SYSTEM DASDAass2_t (* System Configuration *)
  (* Standard: 61499-1 *)
  (* Version 0.4, 2009-03-05, JHC, Holobloc Inc., Deleted Application. *)
  (* Version 0.3, 2003-12-05, JHC, Rockwell Automation, Renamed from NEWSYSTEM. *)
  (* Version 0.2, 2002-11-05, JHC, Rockwell Automation, Fixed missing (empty) FBD in Application. *)
  (* Version 0.1, 2002-01-17, JHC, Rockwell Automation, Minor cleanup *)
  (* Version 0.0, 2000-05-27, JHC, Rockwell Automation *)
  DEVICE HMI_LAYER : FRAME_DEVICE(BOUNDS := [0,0,200,400])
    RESOURCE HMI_1 : PANEL_RESOURCE(COLS := 1, ROWS := 0)
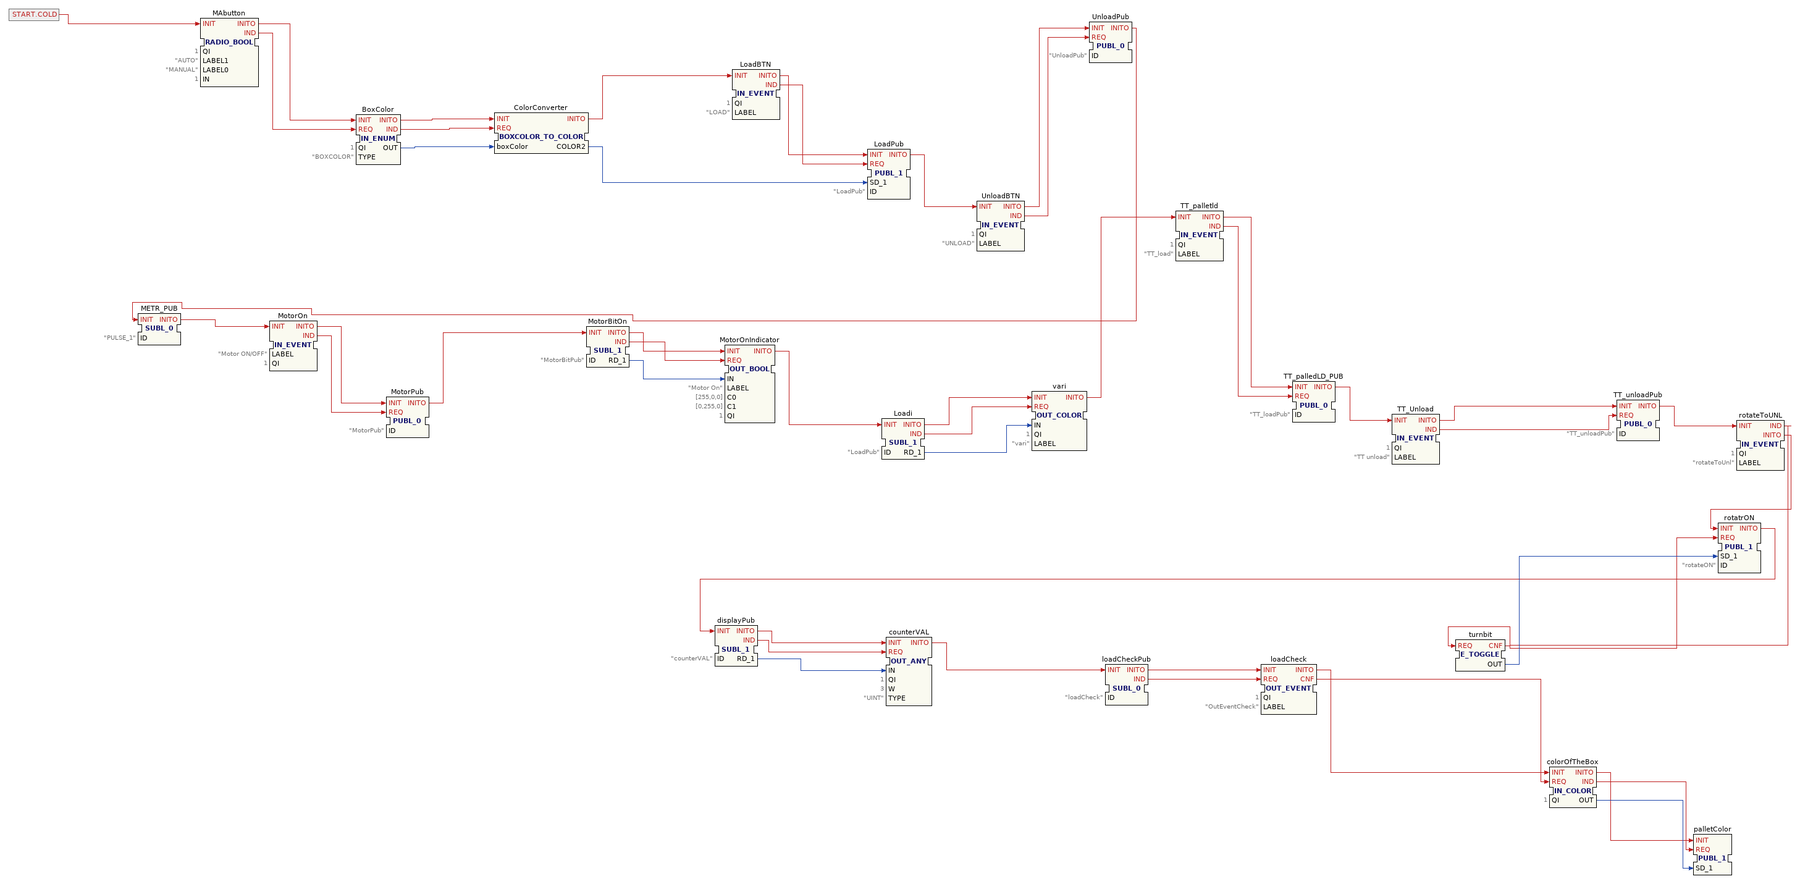
      FBS
        MAbutton : RADIO_BOOL(QI := 1, LABEL1 := "AUTO", LABEL0 := "MANUAL", IN := 1);
        LoadPub : PUBL_1(ID := "LoadPub");
        ColorConverter : BOXCOLOR_TO_COLOR;
        BoxColor : IN_ENUM(QI := 1, TYPE := "BOXCOLOR");
        LoadBTN : IN_EVENT(QI := 1, LABEL := "LOAD");
        Loadi : SUBL_1(ID := "LoadPub");
        vari : OUT_COLOR(QI := 1, LABEL := "vari");
        METR_PUB : SUBL_0(ID := "PULSE_1");
        MotorOn : IN_EVENT(LABEL := "Motor ON/OFF", QI := 1);
        MotorPub : PUBL_0(ID := "MotorPub");
        MotorBitOn : SUBL_1(ID := "MotorBitPub");
        MotorOnIndicator : OUT_BOOL(LABEL := "Motor On", C0 := [255,0,0], C1 := [0,255,0], QI := 1);
        UnloadBTN : IN_EVENT(QI := 1, LABEL := "UNLOAD");
        UnloadPub : PUBL_0(ID := "UnloadPub");
        TT_palletld : IN_EVENT(QI := 1, LABEL := "TT_load");
        TT_palledLD_PUB : PUBL_0(ID := "TT_loadPub");
        displayPub : SUBL_1(ID := "counterVAL");
        counterVAL : OUT_ANY(QI := 1, W := 3, TYPE := "UINT");
        loadCheckPub : SUBL_0(ID := "loadCheck");
        loadCheck : OUT_EVENT(QI := 1, LABEL := "OutEventCheck");
        rotateToUNL : IN_EVENT(QI := 1, LABEL := "rotateToUnl");
        turnbit : E_TOGGLE;
        rotatrON : PUBL_1(ID := "rotateON");
        TT_Unload : IN_EVENT(QI := 1, LABEL := "TT unload");
        TT_unloadPub : PUBL_0(ID := "TT_unloadPub");
        colorOfTheBox : IN_COLOR(QI := 1);
        palletColor : PUBL_1;
      END_FBS
      EVENT_CONNECTIONS
        START.COLD TO MAbutton.INIT;
        BoxColor.INITO TO ColorConverter.INIT;
        BoxColor.IND TO ColorConverter.REQ;
        MAbutton.INITO TO BoxColor.INIT;
        MAbutton.IND TO BoxColor.REQ;
        ColorConverter.INITO TO LoadBTN.INIT;
        LoadBTN.INITO TO LoadPub.INIT;
        LoadBTN.IND TO LoadPub.REQ;
        Loadi.INITO TO vari.INIT;
        Loadi.IND TO vari.REQ;
        METR_PUB.INITO TO MotorOn.INIT;
        MotorOn.INITO TO MotorPub.INIT;
        MotorOn.IND TO MotorPub.REQ;
        MotorPub.INITO TO MotorBitOn.INIT;
        MotorBitOn.INITO TO MotorOnIndicator.INIT;
        MotorBitOn.IND TO MotorOnIndicator.REQ;
        LoadPub.INITO TO UnloadBTN.INIT;
        UnloadBTN.INITO TO UnloadPub.INIT;
        UnloadBTN.IND TO UnloadPub.REQ;
        MotorOnIndicator.INITO TO Loadi.INIT;
        UnloadPub.INITO TO METR_PUB.INIT;
        TT_palletld.INITO TO TT_palledLD_PUB.INIT;
        TT_palletld.IND TO TT_palledLD_PUB.REQ;
        vari.INITO TO TT_palletld.INIT;
        displayPub.INITO TO counterVAL.INIT;
        displayPub.IND TO counterVAL.REQ;
        counterVAL.INITO TO loadCheckPub.INIT;
        loadCheckPub.INITO TO loadCheck.INIT;
        loadCheckPub.IND TO loadCheck.REQ;
        rotateToUNL.IND TO turnbit.REQ;
        rotateToUNL.INITO TO rotatrON.INIT;
        rotatrON.INITO TO displayPub.INIT;
        turnbit.CNF TO rotatrON.REQ;
        TT_palledLD_PUB.INITO TO TT_Unload.INIT;
        TT_Unload.INITO TO TT_unloadPub.INIT;
        TT_unloadPub.INITO TO rotateToUNL.INIT;
        TT_Unload.IND TO TT_unloadPub.REQ;
        loadCheck.INITO TO colorOfTheBox.INIT;
        loadCheck.CNF TO colorOfTheBox.REQ;
        colorOfTheBox.INITO TO palletColor.INIT;
        colorOfTheBox.IND TO palletColor.REQ;
      END_CONNECTIONS
      DATA_CONNECTIONS
        BoxColor.OUT TO ColorConverter.boxColor;
        ColorConverter.COLOR2 TO LoadPub.SD_1;
        Loadi.RD_1 TO vari.IN;
        MotorBitOn.RD_1 TO MotorOnIndicator.IN;
        displayPub.RD_1 TO counterVAL.IN;
        turnbit.OUT TO rotatrON.SD_1;
        colorOfTheBox.OUT TO palletColor.SD_1;
      END_CONNECTIONS
    END_RESOURCE
  END_DEVICE
  DEVICE VIEW_LAYER : FRAME_DEVICE(BOUNDS := [250,0,900,900])
    RESOURCE VIEW_RES : VIEW_PANEL(DIA := 85, SIZE := [10,8], VERTICAL := 0)
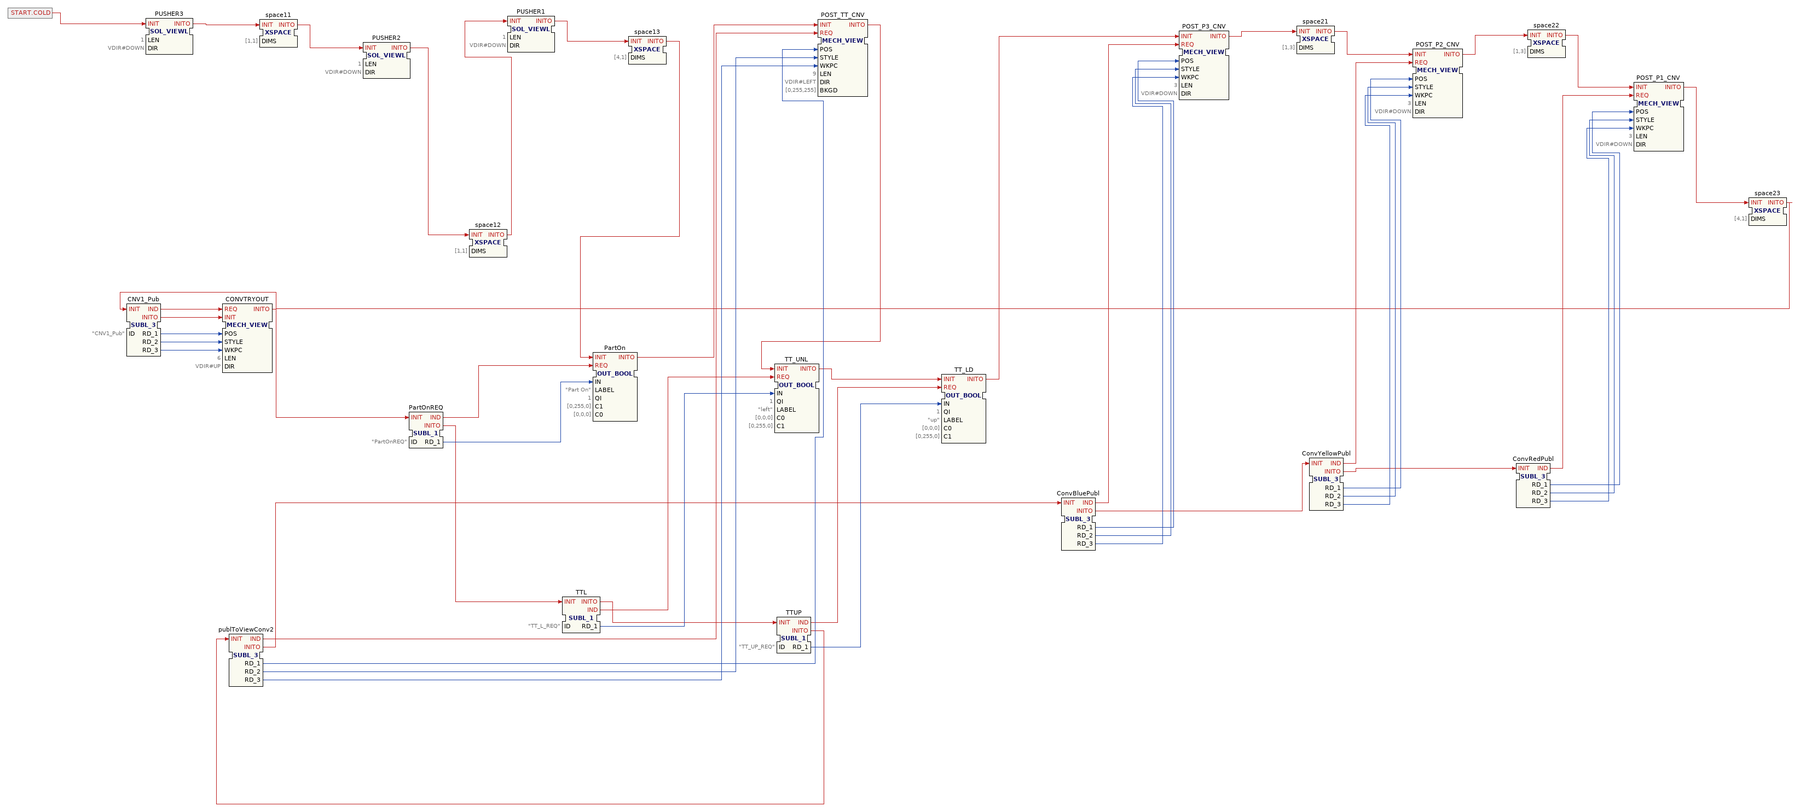
      FBS
        PUSHER3 : SOL_VIEWL(LEN := 1, DIR := VDIR#DOWN);
        space11 : XSPACE(DIMS := [1,1]);
        PUSHER2 : SOL_VIEWL(LEN := 1, DIR := VDIR#DOWN);
        space12 : XSPACE(DIMS := [1,1]);
        PUSHER1 : SOL_VIEWL(LEN := 1, DIR := VDIR#DOWN);
        space13 : XSPACE(DIMS := [4,1]);
        space21 : XSPACE(DIMS := [1,3]);
        space22 : XSPACE(DIMS := [1,3]);
        space23 : XSPACE(DIMS := [4,1]);
        POST_P1_CNV : MECH_VIEW(LEN := 3, DIR := VDIR#DOWN);
        POST_P2_CNV : MECH_VIEW(LEN := 3, DIR := VDIR#DOWN);
        POST_P3_CNV : MECH_VIEW(LEN := 3, DIR := VDIR#DOWN);
        POST_TT_CNV : MECH_VIEW(LEN := 9, DIR := VDIR#LEFT, BKGD := [0,255,255]);
        CONVTRYOUT : MECH_VIEW(LEN := 6, DIR := VDIR#UP);
        CNV1_Pub : SUBL_3(ID := "CNV1_Pub");
        PartOnREQ : SUBL_1(ID := "PartOnREQ");
        PartOn : OUT_BOOL(LABEL := "Part On", QI := 1, C1 := [0,255,0], C0 := [0,0,0]);
        TT_UNL : OUT_BOOL(QI := 1, LABEL := "left", C0 := [0,0,0], C1 := [0,255,0]);
        TT_LD : OUT_BOOL(QI := 1, LABEL := "up", C0 := [0,0,0], C1 := [0,255,0]);
        TTL : SUBL_1(ID := "TT_L_REQ");
        TTUP : SUBL_1(ID := "TT_UP_REQ");
        publToViewConv2 : SUBL_3;
        ConvRedPubl : SUBL_3;
        ConvYellowPubl : SUBL_3;
        ConvBluePubl : SUBL_3;
      END_FBS
      EVENT_CONNECTIONS
        START.COLD TO PUSHER3.INIT;
        PUSHER3.INITO TO space11.INIT;
        space11.INITO TO PUSHER2.INIT;
        PUSHER2.INITO TO space12.INIT;
        space12.INITO TO PUSHER1.INIT;
        PUSHER1.INITO TO space13.INIT;
        space22.INITO TO POST_P1_CNV.INIT;
        POST_P1_CNV.INITO TO space23.INIT;
        space21.INITO TO POST_P2_CNV.INIT;
        POST_P2_CNV.INITO TO space22.INIT;
        POST_P3_CNV.INITO TO space21.INIT;
        CNV1_Pub.IND TO CONVTRYOUT.REQ;
        space23.INITO TO CNV1_Pub.INIT;
        CNV1_Pub.INITO TO CONVTRYOUT.INIT;
        CONVTRYOUT.INITO TO PartOnREQ.INIT;
        space13.INITO TO PartOn.INIT;
        PartOn.INITO TO POST_TT_CNV.INIT;
        PartOnREQ.IND TO PartOn.REQ;
        POST_TT_CNV.INITO TO TT_UNL.INIT;
        TT_UNL.INITO TO TT_LD.INIT;
        TT_LD.INITO TO POST_P3_CNV.INIT;
        PartOnREQ.INITO TO TTL.INIT;
        TTL.INITO TO TTUP.INIT;
        TTL.IND TO TT_UNL.REQ;
        TTUP.IND TO TT_LD.REQ;
        TTUP.INITO TO publToViewConv2.INIT;
        publToViewConv2.IND TO POST_TT_CNV.REQ;
        ConvRedPubl.IND TO POST_P1_CNV.REQ;
        ConvYellowPubl.IND TO POST_P2_CNV.REQ;
        ConvBluePubl.IND TO POST_P3_CNV.REQ;
        publToViewConv2.INITO TO ConvBluePubl.INIT;
        ConvBluePubl.INITO TO ConvYellowPubl.INIT;
        ConvYellowPubl.INITO TO ConvRedPubl.INIT;
      END_CONNECTIONS
      DATA_CONNECTIONS
        CNV1_Pub.RD_1 TO CONVTRYOUT.POS;
        CNV1_Pub.RD_2 TO CONVTRYOUT.STYLE;
        CNV1_Pub.RD_3 TO CONVTRYOUT.WKPC;
        PartOnREQ.RD_1 TO PartOn.IN;
        TTL.RD_1 TO TT_UNL.IN;
        TTUP.RD_1 TO TT_LD.IN;
        publToViewConv2.RD_1 TO POST_TT_CNV.POS;
        publToViewConv2.RD_2 TO POST_TT_CNV.STYLE;
        publToViewConv2.RD_3 TO POST_TT_CNV.WKPC;
        ConvRedPubl.RD_1 TO POST_P1_CNV.POS;
        ConvRedPubl.RD_2 TO POST_P1_CNV.STYLE;
        ConvRedPubl.RD_3 TO POST_P1_CNV.WKPC;
        ConvYellowPubl.RD_1 TO POST_P2_CNV.POS;
        ConvYellowPubl.RD_2 TO POST_P2_CNV.STYLE;
        ConvYellowPubl.RD_3 TO POST_P2_CNV.WKPC;
        ConvBluePubl.RD_1 TO POST_P3_CNV.POS;
        ConvBluePubl.RD_2 TO POST_P3_CNV.STYLE;
        ConvBluePubl.RD_3 TO POST_P3_CNV.WKPC;
      END_CONNECTIONS
    END_RESOURCE
  END_DEVICE
  DEVICE MODEL_LAYER : FRAME_DEVICE
    RESOURCE INIT_CLOCK : PANEL_RESOURCE
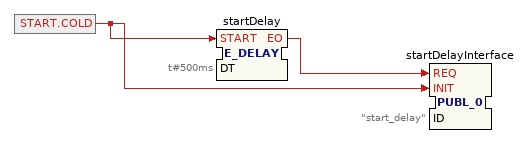
      FBS
        startDelay : E_DELAY(DT := t#500ms);
        startDelayInterface : PUBL_0(ID := "start_delay");
      END_FBS
      EVENT_CONNECTIONS
        START.COLD TO startDelay.START;
        startDelay.EO TO startDelayInterface.REQ;
        START.COLD TO startDelayInterface.INIT;
      END_CONNECTIONS
    END_RESOURCE
    RESOURCE MODEL_CLOCK : PANEL_RESOURCE
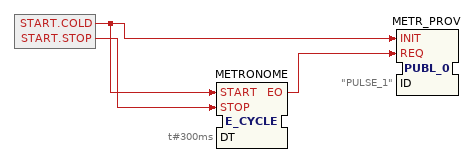
      FBS
        METRONOME : E_CYCLE(DT := t#300ms);
        METR_PROV : PUBL_0(ID := "PULSE_1");
      END_FBS
      EVENT_CONNECTIONS
        START.COLD TO METRONOME.START;
        START.STOP TO METRONOME.STOP;
        START.COLD TO METR_PROV.INIT;
        METRONOME.EO TO METR_PROV.REQ;
      END_CONNECTIONS
    END_RESOURCE
    RESOURCE CNV_1_MODEL : PANEL_RESOURCE
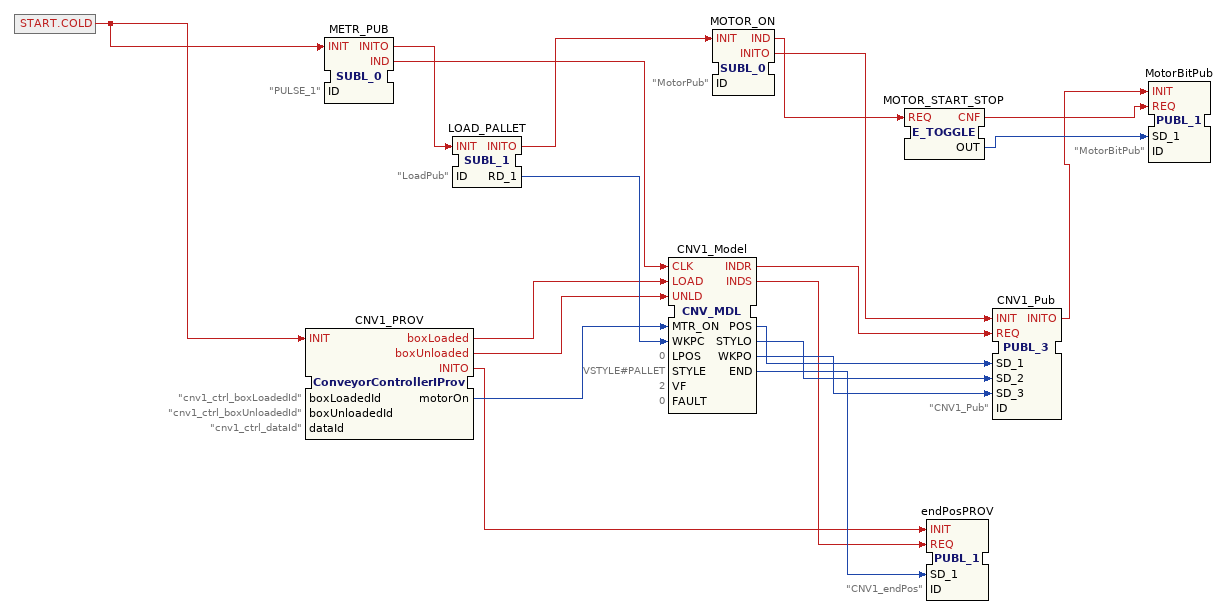
      FBS
        METR_PUB : SUBL_0(ID := "PULSE_1");
        MOTOR_ON : SUBL_0(ID := "MotorPub");
        LOAD_PALLET : SUBL_1(ID := "LoadPub");
        MOTOR_START_STOP : E_TOGGLE;
        CNV1_Model : CNV_MDL(LPOS := 0, STYLE := VSTYLE#PALLET, VF := 2, FAULT := 0);
        CNV1_Pub : PUBL_3(ID := "CNV1_Pub");
        MotorBitPub : PUBL_1(ID := "MotorBitPub");
        endPosPROV : PUBL_1(ID := "CNV1_endPos");
        CNV1_PROV : ConveyorControllerIProv(boxLoadedId := "cnv1_ctrl_boxLoadedId", boxUnloadedId := "cnv1_ctrl_boxUnloadedId", dataId := "cnv1_ctrl_dataId");
      END_FBS
      EVENT_CONNECTIONS
        START.COLD TO METR_PUB.INIT;
        METR_PUB.INITO TO LOAD_PALLET.INIT;
        LOAD_PALLET.INITO TO MOTOR_ON.INIT;
        MOTOR_ON.IND TO MOTOR_START_STOP.REQ;
        METR_PUB.IND TO CNV1_Model.CLK;
        MOTOR_ON.INITO TO CNV1_Pub.INIT;
        CNV1_Model.INDR TO CNV1_Pub.REQ;
        CNV1_Pub.INITO TO MotorBitPub.INIT;
        MOTOR_START_STOP.CNF TO MotorBitPub.REQ;
        CNV1_PROV.boxLoaded TO CNV1_Model.LOAD;
        CNV1_PROV.boxUnloaded TO CNV1_Model.UNLD;
        START.COLD TO CNV1_PROV.INIT;
        CNV1_PROV.INITO TO endPosPROV.INIT;
        CNV1_Model.INDS TO endPosPROV.REQ;
      END_CONNECTIONS
      DATA_CONNECTIONS
        CNV1_Model.POS TO CNV1_Pub.SD_1;
        CNV1_Model.STYLO TO CNV1_Pub.SD_2;
        CNV1_Model.WKPO TO CNV1_Pub.SD_3;
        MOTOR_START_STOP.OUT TO MotorBitPub.SD_1;
        CNV1_Model.END TO endPosPROV.SD_1;
        CNV1_PROV.motorOn TO CNV1_Model.MTR_ON;
        LOAD_PALLET.RD_1 TO CNV1_Model.WKPC;
      END_CONNECTIONS
    END_RESOURCE
    RESOURCE TT_MODEL : PANEL_RESOURCE
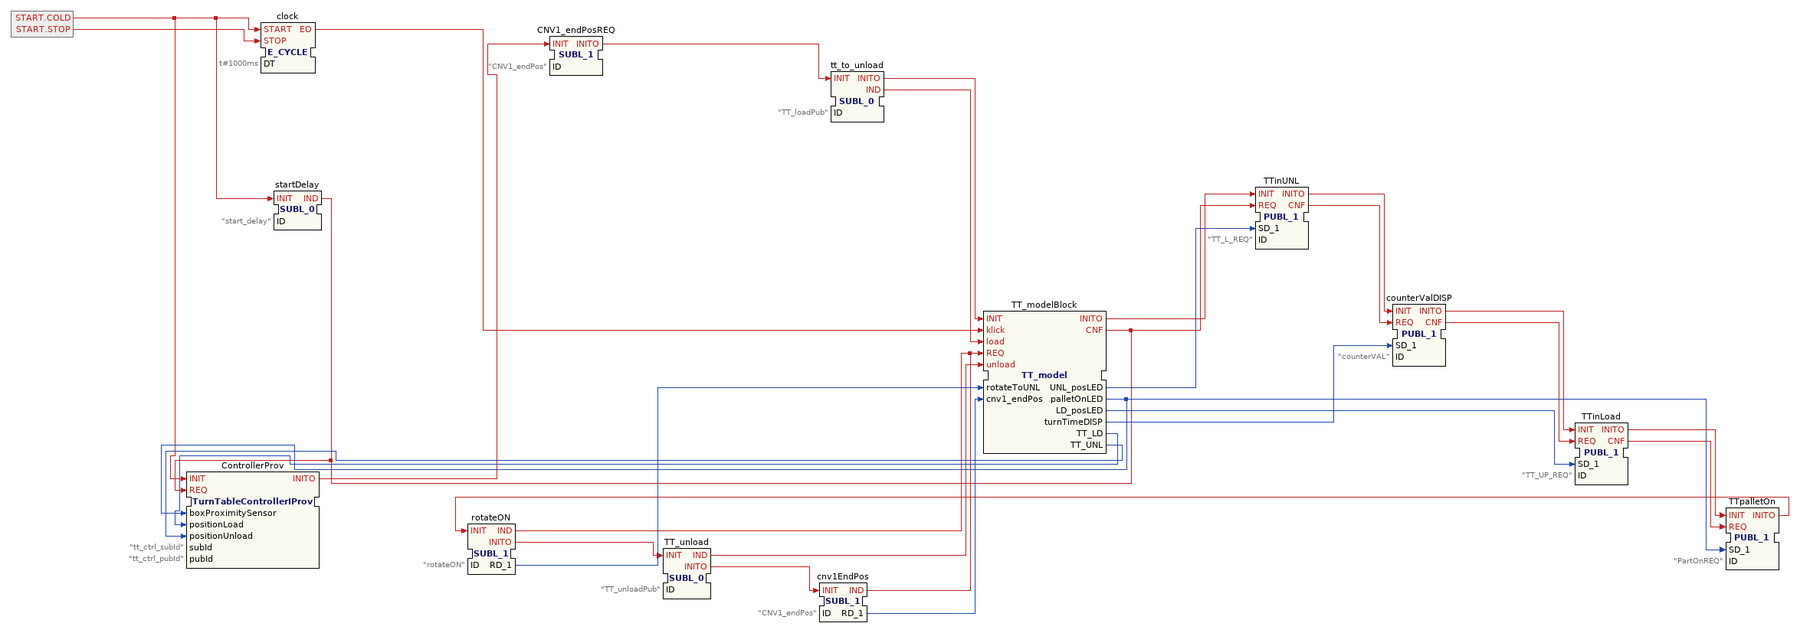
      FBS
        CNV1_endPosREQ : SUBL_1(ID := "CNV1_endPos");
        clock : E_CYCLE(DT := t#1000ms);
        ControllerProv : TurnTableControllerIProv(subId := "tt_ctrl_subId", pubId := "tt_ctrl_pubId");
        TTinUNL : PUBL_1(ID := "TT_L_REQ");
        tt_to_unload : SUBL_0(ID := "TT_loadPub");
        counterValDISP : PUBL_1(ID := "counterVAL");
        TTinLoad : PUBL_1(ID := "TT_UP_REQ");
        TTpalletOn : PUBL_1(ID := "PartOnREQ");
        rotateON : SUBL_1(ID := "rotateON");
        TT_modelBlock : TT_model;
        TT_unload : SUBL_0(ID := "TT_unloadPub");
        startDelay : SUBL_0(ID := "start_delay");
        cnv1EndPos : SUBL_1(ID := "CNV1_endPos");
      END_FBS
      EVENT_CONNECTIONS
        START.COLD TO clock.START;
        START.STOP TO clock.STOP;
        START.COLD TO ControllerProv.INIT;
        ControllerProv.INITO TO CNV1_endPosREQ.INIT;
        CNV1_endPosREQ.INITO TO tt_to_unload.INIT;
        TTinUNL.INITO TO counterValDISP.INIT;
        TTinUNL.CNF TO counterValDISP.REQ;
        counterValDISP.INITO TO TTinLoad.INIT;
        counterValDISP.CNF TO TTinLoad.REQ;
        TTinLoad.INITO TO TTpalletOn.INIT;
        TTinLoad.CNF TO TTpalletOn.REQ;
        TTpalletOn.INITO TO rotateON.INIT;
        tt_to_unload.INITO TO TT_modelBlock.INIT;
        TT_modelBlock.INITO TO TTinUNL.INIT;
        TT_modelBlock.CNF TO TTinUNL.REQ;
        clock.EO TO TT_modelBlock.klick;
        tt_to_unload.IND TO TT_modelBlock.load;
        rotateON.IND TO TT_modelBlock.REQ;
        rotateON.INITO TO TT_unload.INIT;
        TT_unload.IND TO TT_modelBlock.unload;
        START.COLD TO startDelay.INIT;
        startDelay.IND TO ControllerProv.REQ;
        TT_modelBlock.CNF TO ControllerProv.REQ;
        TT_unload.INITO TO cnv1EndPos.INIT;
        cnv1EndPos.IND TO TT_modelBlock.REQ;
      END_CONNECTIONS
      DATA_CONNECTIONS
        TT_modelBlock.UNL_posLED TO TTinUNL.SD_1;
        TT_modelBlock.palletOnLED TO TTpalletOn.SD_1;
        TT_modelBlock.LD_posLED TO TTinLoad.SD_1;
        TT_modelBlock.turnTimeDISP TO counterValDISP.SD_1;
        TT_modelBlock.palletOnLED TO ControllerProv.boxProximitySensor;
        rotateON.RD_1 TO TT_modelBlock.rotateToUNL;
        TT_modelBlock.TT_LD TO ControllerProv.positionLoad;
        TT_modelBlock.TT_UNL TO ControllerProv.positionUnload;
        cnv1EndPos.RD_1 TO TT_modelBlock.cnv1_endPos;
      END_CONNECTIONS
    END_RESOURCE
    RESOURCE CNV_2_MODEL : PANEL_RESOURCE
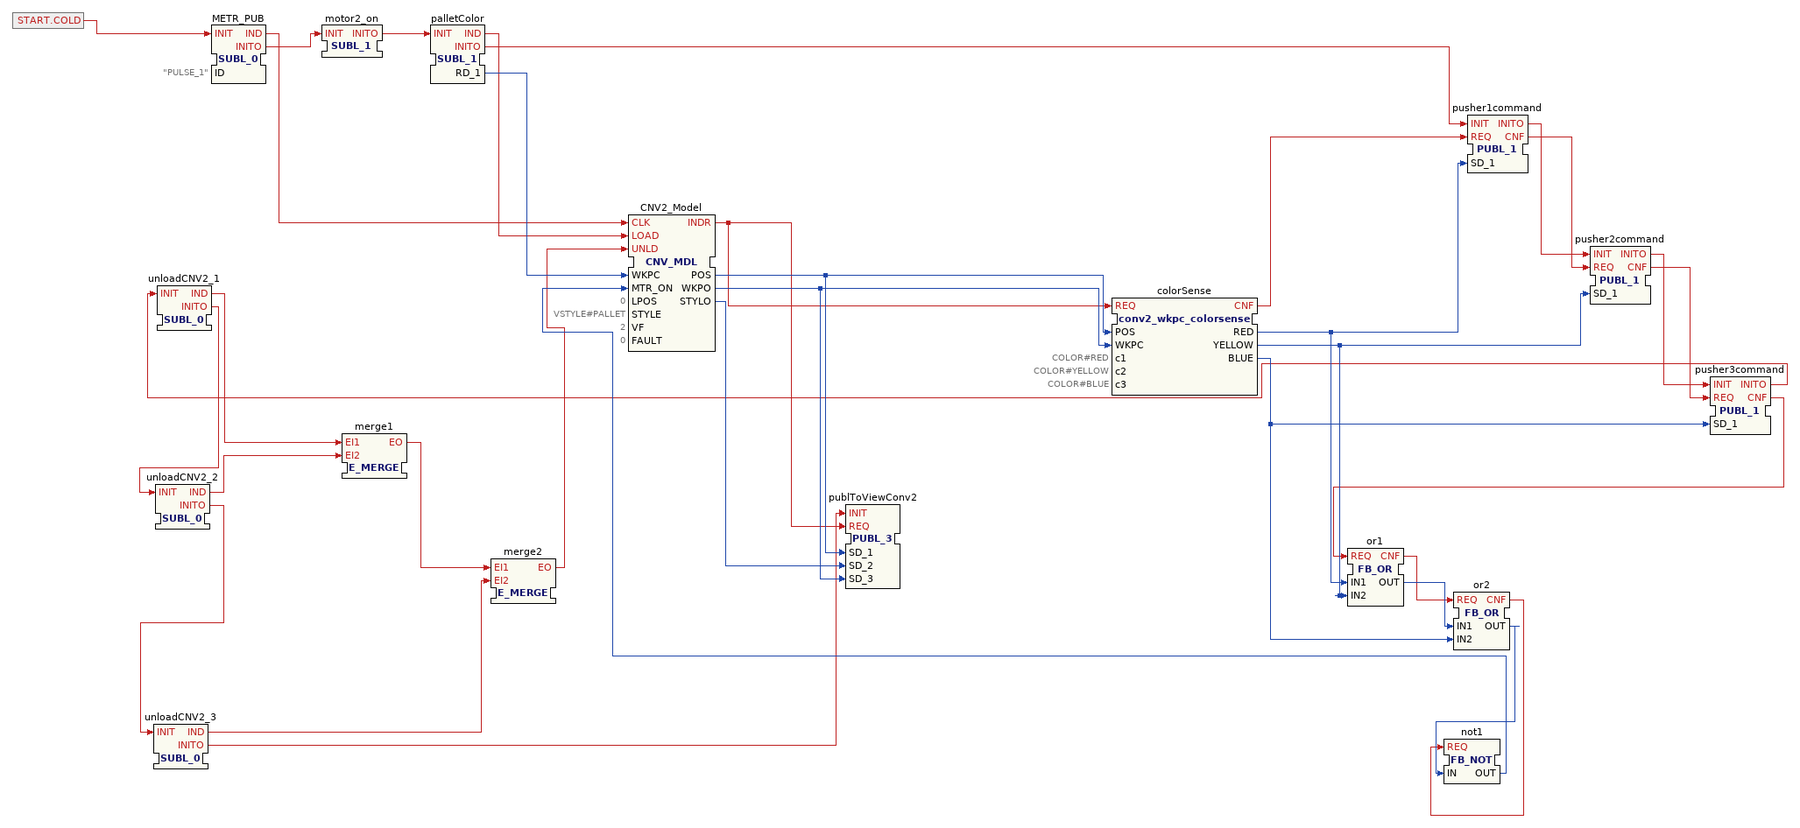
      FBS
        CNV2_Model : CNV_MDL(LPOS := 0, STYLE := VSTYLE#PALLET, VF := 2, FAULT := 0);
        METR_PUB : SUBL_0(ID := "PULSE_1");
        palletColor : SUBL_1;
        motor2_on : SUBL_1;
        colorSense : conv2_wkpc_colorsense(c1 := COLOR#RED, c2 := COLOR#YELLOW, c3 := COLOR#BLUE);
        pusher1command : PUBL_1;
        pusher2command : PUBL_1;
        pusher3command : PUBL_1;
        unloadCNV2_1 : SUBL_0;
        merge1 : E_MERGE;
        merge2 : E_MERGE;
        unloadCNV2_2 : SUBL_0;
        unloadCNV2_3 : SUBL_0;
        or1 : FB_OR;
        or2 : FB_OR;
        not1 : FB_NOT;
        publToViewConv2 : PUBL_3;
      END_FBS
      EVENT_CONNECTIONS
        START.COLD TO METR_PUB.INIT;
        METR_PUB.IND TO CNV2_Model.CLK;
        palletColor.IND TO CNV2_Model.LOAD;
        METR_PUB.INITO TO motor2_on.INIT;
        motor2_on.INITO TO palletColor.INIT;
        palletColor.INITO TO pusher1command.INIT;
        pusher1command.INITO TO pusher2command.INIT;
        pusher2command.INITO TO pusher3command.INIT;
        colorSense.CNF TO pusher1command.REQ;
        pusher1command.CNF TO pusher2command.REQ;
        pusher2command.CNF TO pusher3command.REQ;
        pusher3command.INITO TO unloadCNV2_1.INIT;
        unloadCNV2_1.IND TO merge1.EI1;
        merge1.EO TO merge2.EI1;
        unloadCNV2_1.INITO TO unloadCNV2_2.INIT;
        unloadCNV2_2.IND TO merge1.EI2;
        unloadCNV2_2.INITO TO unloadCNV2_3.INIT;
        unloadCNV2_3.IND TO merge2.EI2;
        merge2.EO TO CNV2_Model.UNLD;
        pusher3command.CNF TO or1.REQ;
        or1.CNF TO or2.REQ;
        or2.CNF TO not1.REQ;
        unloadCNV2_3.INITO TO publToViewConv2.INIT;
        CNV2_Model.INDR TO publToViewConv2.REQ;
        CNV2_Model.INDR TO colorSense.REQ;
      END_CONNECTIONS
      DATA_CONNECTIONS
        palletColor.RD_1 TO CNV2_Model.WKPC;
        CNV2_Model.POS TO colorSense.POS;
        CNV2_Model.WKPO TO colorSense.WKPC;
        colorSense.RED TO pusher1command.SD_1;
        colorSense.YELLOW TO pusher2command.SD_1;
        colorSense.BLUE TO pusher3command.SD_1;
        colorSense.RED TO or1.IN1;
        colorSense.YELLOW TO or1.IN2;
        or1.OUT TO or2.IN1;
        colorSense.BLUE TO or2.IN2;
        or2.OUT TO not1.IN;
        not1.OUT TO CNV2_Model.MTR_ON;
        CNV2_Model.POS TO publToViewConv2.SD_1;
        CNV2_Model.STYLO TO publToViewConv2.SD_2;
        CNV2_Model.WKPO TO publToViewConv2.SD_3;
      END_CONNECTIONS
    END_RESOURCE
    RESOURCE PUSHER1_MODEL : PANEL_RESOURCE
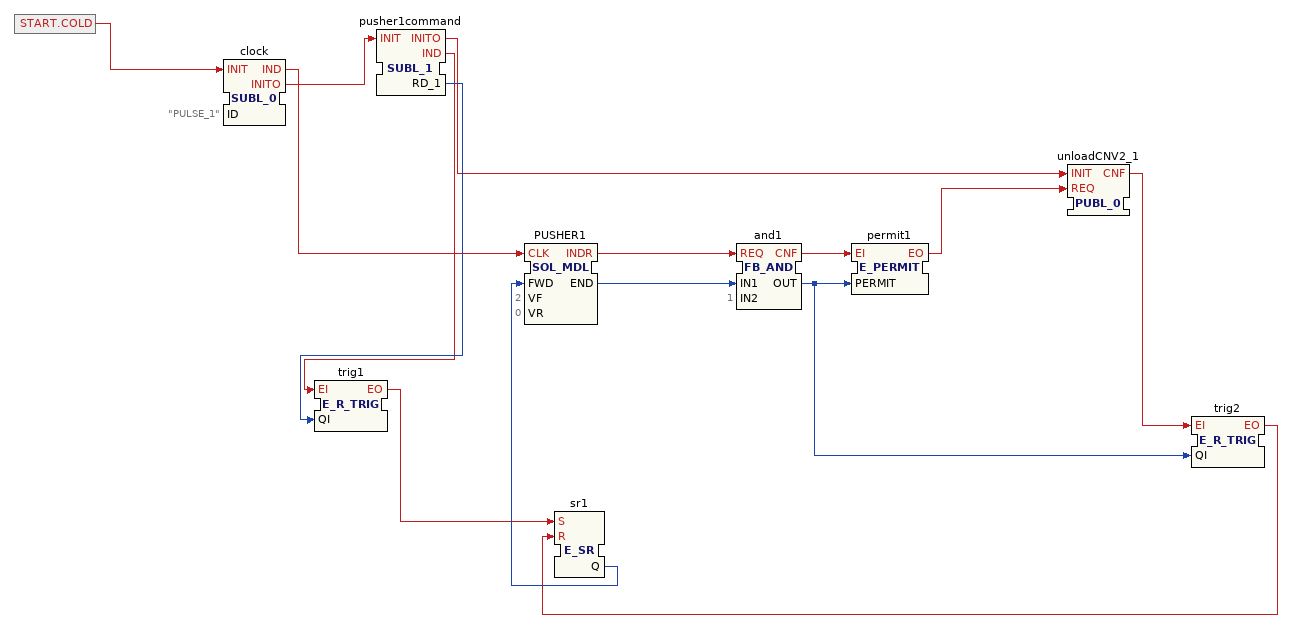
      FBS
        PUSHER1 : SOL_MDL(VF := 2, VR := 0);
        clock : SUBL_0(ID := "PULSE_1");
        pusher1command : SUBL_1;
        and1 : FB_AND(IN2 := 1);
        permit1 : E_PERMIT;
        unloadCNV2_1 : PUBL_0;
        trig1 : E_R_TRIG;
        trig2 : E_R_TRIG;
        sr1 : E_SR;
      END_FBS
      EVENT_CONNECTIONS
        START.COLD TO clock.INIT;
        clock.IND TO PUSHER1.CLK;
        clock.INITO TO pusher1command.INIT;
        PUSHER1.INDR TO and1.REQ;
        and1.CNF TO permit1.EI;
        pusher1command.INITO TO unloadCNV2_1.INIT;
        permit1.EO TO unloadCNV2_1.REQ;
        unloadCNV2_1.CNF TO trig2.EI;
        pusher1command.IND TO trig1.EI;
        trig1.EO TO sr1.S;
        trig2.EO TO sr1.R;
      END_CONNECTIONS
      DATA_CONNECTIONS
        PUSHER1.END TO and1.IN1;
        and1.OUT TO permit1.PERMIT;
        pusher1command.RD_1 TO trig1.QI;
        and1.OUT TO trig2.QI;
        sr1.Q TO PUSHER1.FWD;
      END_CONNECTIONS
    END_RESOURCE
    RESOURCE PUSHER2_MODEL : PANEL_RESOURCE
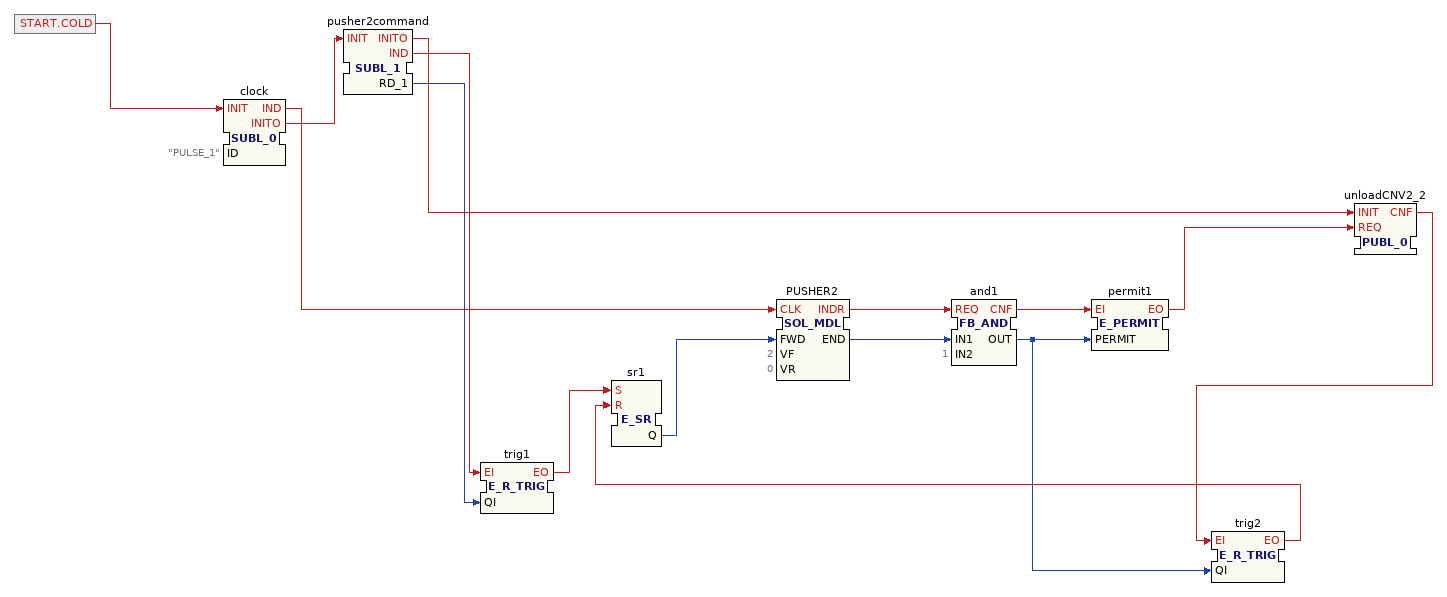
      FBS
        PUSHER2 : SOL_MDL(VF := 2, VR := 0);
        clock : SUBL_0(ID := "PULSE_1");
        pusher2command : SUBL_1;
        and1 : FB_AND(IN2 := 1);
        permit1 : E_PERMIT;
        unloadCNV2_2 : PUBL_0;
        sr1 : E_SR;
        trig1 : E_R_TRIG;
        trig2 : E_R_TRIG;
      END_FBS
      EVENT_CONNECTIONS
        START.COLD TO clock.INIT;
        clock.IND TO PUSHER2.CLK;
        clock.INITO TO pusher2command.INIT;
        PUSHER2.INDR TO and1.REQ;
        and1.CNF TO permit1.EI;
        pusher2command.INITO TO unloadCNV2_2.INIT;
        permit1.EO TO unloadCNV2_2.REQ;
        pusher2command.IND TO trig1.EI;
        trig1.EO TO sr1.S;
        unloadCNV2_2.CNF TO trig2.EI;
        trig2.EO TO sr1.R;
      END_CONNECTIONS
      DATA_CONNECTIONS
        PUSHER2.END TO and1.IN1;
        and1.OUT TO permit1.PERMIT;
        pusher2command.RD_1 TO trig1.QI;
        and1.OUT TO trig2.QI;
        sr1.Q TO PUSHER2.FWD;
      END_CONNECTIONS
    END_RESOURCE
    RESOURCE PUSHER3_MODEL : PANEL_RESOURCE
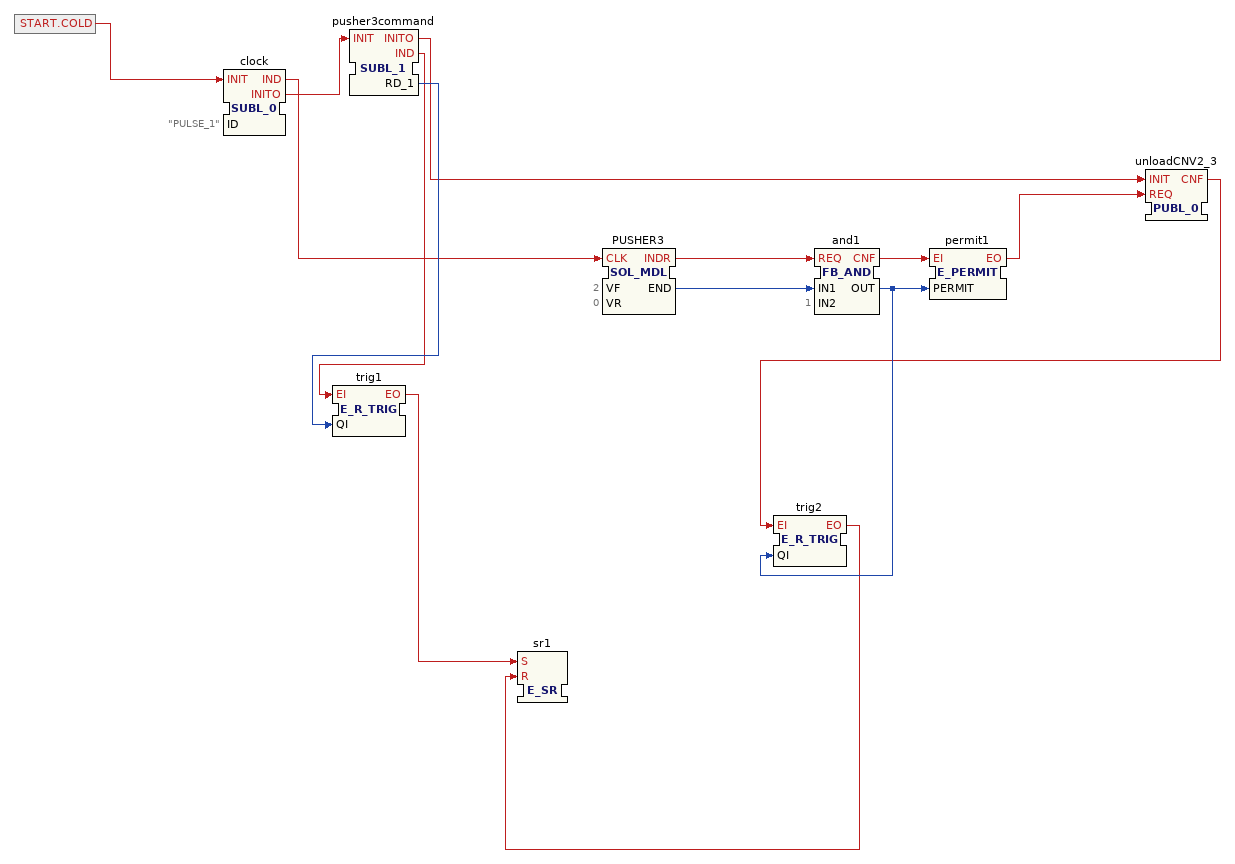
      FBS
        PUSHER3 : SOL_MDL(VF := 2, VR := 0);
        clock : SUBL_0(ID := "PULSE_1");
        pusher3command : SUBL_1;
        and1 : FB_AND(IN2 := 1);
        permit1 : E_PERMIT;
        unloadCNV2_3 : PUBL_0;
        trig1 : E_R_TRIG;
        trig2 : E_R_TRIG;
        sr1 : E_SR;
      END_FBS
      EVENT_CONNECTIONS
        START.COLD TO clock.INIT;
        clock.IND TO PUSHER3.CLK;
        clock.INITO TO pusher3command.INIT;
        PUSHER3.INDR TO and1.REQ;
        and1.CNF TO permit1.EI;
        pusher3command.INITO TO unloadCNV2_3.INIT;
        permit1.EO TO unloadCNV2_3.REQ;
        pusher3command.IND TO trig1.EI;
        trig1.EO TO sr1.S;
        unloadCNV2_3.CNF TO trig2.EI;
        trig2.EO TO sr1.R;
      END_CONNECTIONS
      DATA_CONNECTIONS
        PUSHER3.END TO and1.IN1;
        and1.OUT TO permit1.PERMIT;
        pusher3command.RD_1 TO trig1.QI;
        and1.OUT TO trig2.QI;
      END_CONNECTIONS
    END_RESOURCE
    RESOURCE CONVred_MODEL : PANEL_RESOURCE
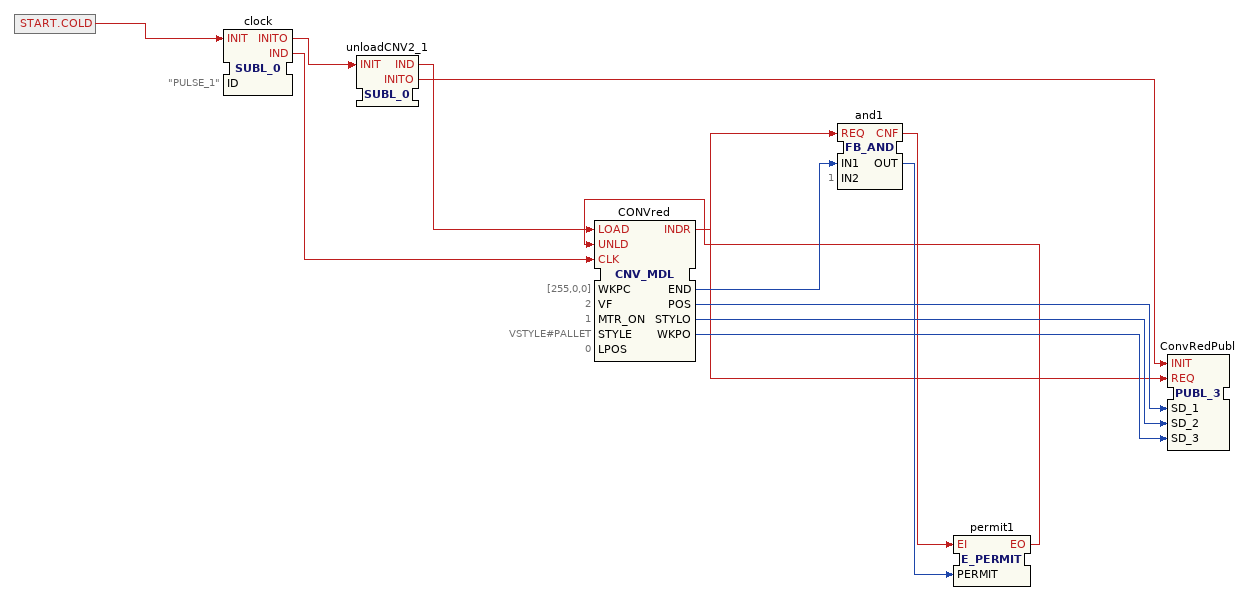
      FBS
        unloadCNV2_1 : SUBL_0;
        CONVred : CNV_MDL(WKPC := [255,0,0], VF := 2, MTR_ON := 1, STYLE := VSTYLE#PALLET, LPOS := 0);
        and1 : FB_AND(IN2 := 1);
        permit1 : E_PERMIT;
        ConvRedPubl : PUBL_3;
        clock : SUBL_0(ID := "PULSE_1");
      END_FBS
      EVENT_CONNECTIONS
        unloadCNV2_1.IND TO CONVred.LOAD;
        and1.CNF TO permit1.EI;
        permit1.EO TO CONVred.UNLD;
        unloadCNV2_1.INITO TO ConvRedPubl.INIT;
        CONVred.INDR TO ConvRedPubl.REQ;
        START.COLD TO clock.INIT;
        clock.INITO TO unloadCNV2_1.INIT;
        clock.IND TO CONVred.CLK;
        CONVred.INDR TO and1.REQ;
      END_CONNECTIONS
      DATA_CONNECTIONS
        CONVred.END TO and1.IN1;
        and1.OUT TO permit1.PERMIT;
        CONVred.POS TO ConvRedPubl.SD_1;
        CONVred.STYLO TO ConvRedPubl.SD_2;
        CONVred.WKPO TO ConvRedPubl.SD_3;
      END_CONNECTIONS
    END_RESOURCE
    RESOURCE CONVyellow_MODEL : PANEL_RESOURCE
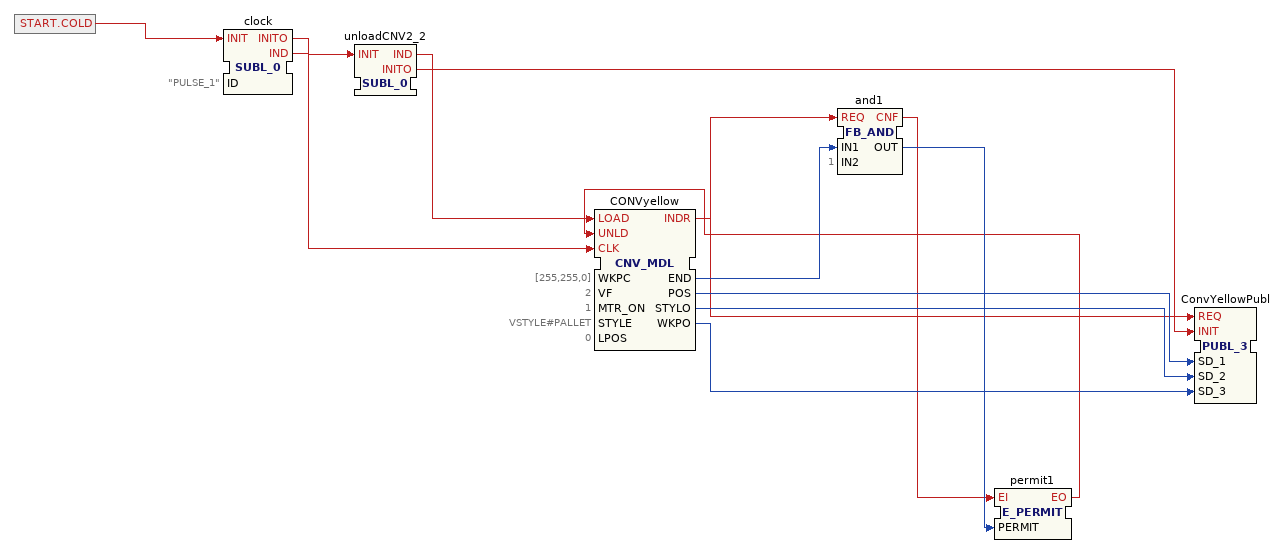
      FBS
        unloadCNV2_2 : SUBL_0;
        CONVyellow : CNV_MDL(WKPC := [255,255,0], VF := 2, MTR_ON := 1, STYLE := VSTYLE#PALLET, LPOS := 0);
        and1 : FB_AND(IN2 := 1);
        permit1 : E_PERMIT;
        ConvYellowPubl : PUBL_3;
        clock : SUBL_0(ID := "PULSE_1");
      END_FBS
      EVENT_CONNECTIONS
        unloadCNV2_2.IND TO CONVyellow.LOAD;
        and1.CNF TO permit1.EI;
        permit1.EO TO CONVyellow.UNLD;
        CONVyellow.INDR TO ConvYellowPubl.REQ;
        unloadCNV2_2.INITO TO ConvYellowPubl.INIT;
        START.COLD TO clock.INIT;
        clock.INITO TO unloadCNV2_2.INIT;
        clock.IND TO CONVyellow.CLK;
        CONVyellow.INDR TO and1.REQ;
      END_CONNECTIONS
      DATA_CONNECTIONS
        CONVyellow.END TO and1.IN1;
        and1.OUT TO permit1.PERMIT;
        CONVyellow.POS TO ConvYellowPubl.SD_1;
        CONVyellow.STYLO TO ConvYellowPubl.SD_2;
        CONVyellow.WKPO TO ConvYellowPubl.SD_3;
      END_CONNECTIONS
    END_RESOURCE
    RESOURCE CONVblue_MODEL : PANEL_RESOURCE
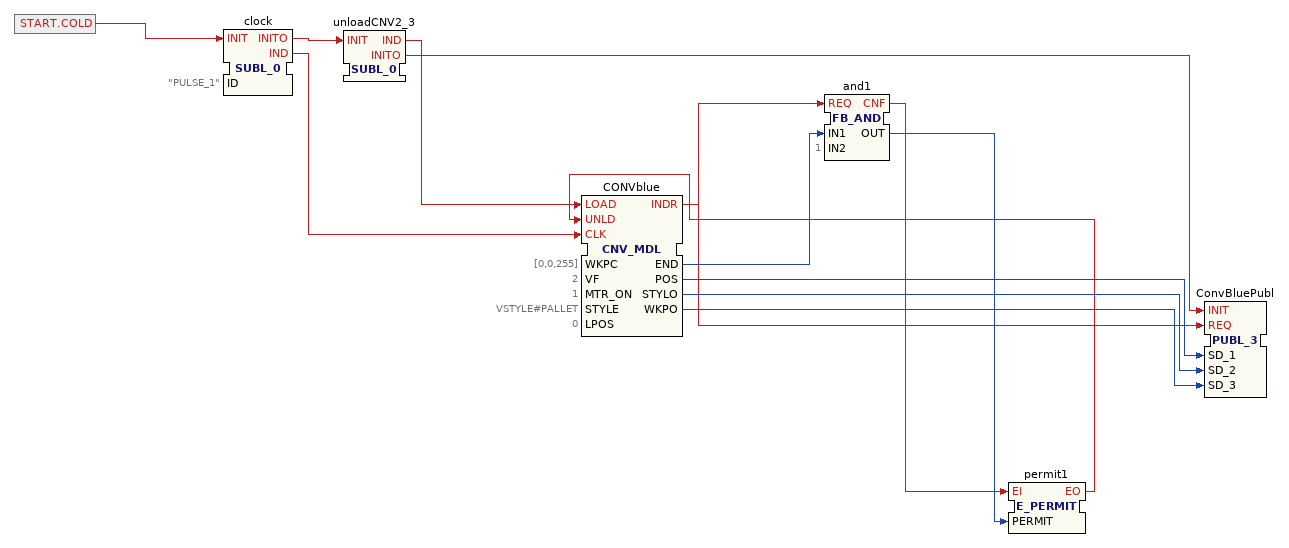
      FBS
        unloadCNV2_3 : SUBL_0;
        CONVblue : CNV_MDL(WKPC := [0,0,255], VF := 2, MTR_ON := 1, STYLE := VSTYLE#PALLET, LPOS := 0);
        and1 : FB_AND(IN2 := 1);
        permit1 : E_PERMIT;
        ConvBluePubl : PUBL_3;
        clock : SUBL_0(ID := "PULSE_1");
      END_FBS
      EVENT_CONNECTIONS
        unloadCNV2_3.IND TO CONVblue.LOAD;
        and1.CNF TO permit1.EI;
        permit1.EO TO CONVblue.UNLD;
        unloadCNV2_3.INITO TO ConvBluePubl.INIT;
        CONVblue.INDR TO ConvBluePubl.REQ;
        START.COLD TO clock.INIT;
        clock.INITO TO unloadCNV2_3.INIT;
        clock.IND TO CONVblue.CLK;
        CONVblue.INDR TO and1.REQ;
      END_CONNECTIONS
      DATA_CONNECTIONS
        CONVblue.END TO and1.IN1;
        and1.OUT TO permit1.PERMIT;
        CONVblue.POS TO ConvBluePubl.SD_1;
        CONVblue.STYLO TO ConvBluePubl.SD_2;
        CONVblue.WKPO TO ConvBluePubl.SD_3;
      END_CONNECTIONS
    END_RESOURCE
  END_DEVICE
  DEVICE CONTROLLER_LAYER : FRAME_DEVICE(BOUNDS := [0,400,200,200])
    RESOURCE Conveyor1Controller : PANEL_RESOURCE(ROWS := 0, COLS := 1)
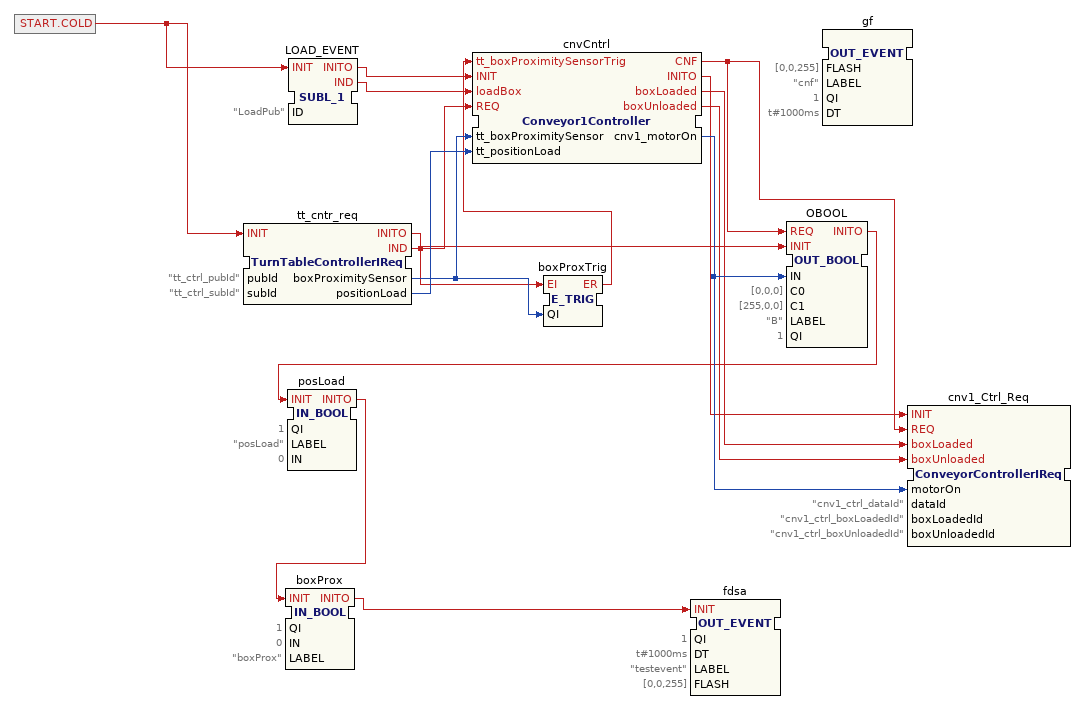
      FBS
        OBOOL : OUT_BOOL(C0 := [0,0,0], C1 := [255,0,0], LABEL := "B", QI := 1);
        gf : OUT_EVENT(FLASH := [0,0,255], LABEL := "cnf", QI := 1, DT := t#1000ms);
        cnvCntrl : Conveyor1Controller;
        boxProxTrig : E_TRIG;
        fdsa : OUT_EVENT(QI := 1, DT := t#1000ms, LABEL := "testevent", FLASH := [0,0,255]);
        posLoad : IN_BOOL(QI := 1, LABEL := "posLoad", IN := 0);
        boxProx : IN_BOOL(QI := 1, IN := 0, LABEL := "boxProx");
        cnv1_Ctrl_Req : ConveyorControllerIReq(dataId := "cnv1_ctrl_dataId", boxLoadedId := "cnv1_ctrl_boxLoadedId", boxUnloadedId := "cnv1_ctrl_boxUnloadedId");
        LOAD_EVENT : SUBL_1(ID := "LoadPub");
        tt_cntr_req : TurnTableControllerIReq(pubId := "tt_ctrl_pubId", subId := "tt_ctrl_subId");
      END_FBS
      EVENT_CONNECTIONS
        cnvCntrl.CNF TO OBOOL.REQ;
        posLoad.INITO TO boxProx.INIT;
        boxProx.INITO TO fdsa.INIT;
        boxProxTrig.ER TO cnvCntrl.tt_boxProximitySensorTrig;
        cnvCntrl.INITO TO cnv1_Ctrl_Req.INIT;
        cnvCntrl.CNF TO cnv1_Ctrl_Req.REQ;
        cnvCntrl.boxLoaded TO cnv1_Ctrl_Req.boxLoaded;
        cnvCntrl.boxUnloaded TO cnv1_Ctrl_Req.boxUnloaded;
        START.COLD TO LOAD_EVENT.INIT;
        LOAD_EVENT.INITO TO cnvCntrl.INIT;
        LOAD_EVENT.IND TO cnvCntrl.loadBox;
        START.COLD TO tt_cntr_req.INIT;
        tt_cntr_req.INITO TO OBOOL.INIT;
        OBOOL.INITO TO posLoad.INIT;
        tt_cntr_req.IND TO cnvCntrl.REQ;
        tt_cntr_req.IND TO boxProxTrig.EI;
      END_CONNECTIONS
      DATA_CONNECTIONS
        cnvCntrl.cnv1_motorOn TO OBOOL.IN;
        cnvCntrl.cnv1_motorOn TO cnv1_Ctrl_Req.motorOn;
        tt_cntr_req.boxProximitySensor TO cnvCntrl.tt_boxProximitySensor;
        tt_cntr_req.boxProximitySensor TO boxProxTrig.QI;
        tt_cntr_req.positionLoad TO cnvCntrl.tt_positionLoad;
      END_CONNECTIONS
    END_RESOURCE
  END_DEVICE
END_SYSTEM
